Fanuc KAREL source: kt00979.KL

PROGRAM KT00979
%STACKSIZE=65535
%PRIORITY=65535
%NOLOCKGROUP
VAR
I1 : INTEGER
I2 : INTEGER
OUT : POSITION
-- UNRESOLVED DECLARATIONS (source type spelling not recovered)
-- CFG : TYPE_0x001C (type_u16=0x001C)
BEGIN
I1=2
I2=3
I1=2
I2=3
-- UNRESOLVED_PC line 13 opcodes [9D 22 A5] marker_code=64
-- UNRESOLVED_PC line 14 opcodes [27 27 21 64 27 21 64 27 21 64 27 21 64 27 21 64 27 21 64 22 76 7E 4A] marker_code=79
END KT00979
